# EPICS autosave request: BPMApp/Db/BPMFmcPico1m_4ch_settings.req
$(P)$(R)FMCPICORngR0
$(P)$(R)FMCPICORngR1
$(P)$(R)FMCPICORngR2
$(P)$(R)FMCPICORngR3
